DATA_BLOCK "ModeDB"
{ S7_Optimized_Access := 'FALSE' }
VERSION : 0.1
NON_RETAIN
   STRUCT
      Gen : "ModeGenStruct";
   END_STRUCT;


BEGIN

END_DATA_BLOCK

